Staubli VAL3: pantalla.pgx

program pantalla()
begin
  userPage(sMonitor)
  cls(sMonitor)
  title(sMonitor, "Start to recicling")
  gotoxy(sMonitor, 35,13)
  put(sMonitor, "EXIT")
  do
    gotoxy(sMonitor, 0,1)
    put(sMonitor, "Port 1102:")
    gotoxy(sMonitor, 12,1)
    switch nConnection
      case -1
        put(sMonitor, "Waiting connection")
      break
      case 1
        put(sMonitor, "Connected succesful")
        putln(sMonitor,"Go to bin: ")
        switch nRecvData
          case 48
            put(sMonitor, "Yellow")
          break
          case 49
           put(sMonitor, "Blue")
          break
        case 50
          put(sMonitor, "Green")
        break
        case 51
          put(sMonitor, "Brown")
        break
        default
          putln(sMonitor, "Bin selected no correct")
        break
      endSwitch
      break
      default
        put(sMonitor, "Connection lose")
      break
    endSwitch
  until 1==1
end
